// TIA Portal V20 export
DATA_BLOCK "Data_to_Safety"   // DB3
{ S7_Optimized_Access := 'TRUE' }
// stored: MemoryReserve 100
   VAR
      rcv_buffer : Array[0..121] of Byte;
      rcv_buffer2 : Array[0..121] of Byte;
   END_VAR
BEGIN
END_DATA_BLOCK
